{attribute 'qualified_only'}
{attribute 'strict'}
TYPE E_AlarmState :
(
	OFF := 0,
	LEVEL_SENSOR,
	BOTTLE_SENSOR,
	CONVEYER
	
);
END_TYPE

(* stored: Version 1.1.0.1, ProductVersion 3.1.4024.16
   DUT E_AlarmState: Id {c07ba835-0eff-418e-87a4-e3c136acc91e} *)
